METHOD PROTECTED T22_TestAddRecipeFromTemplate
VAR
	bResult: BOOL;
	sttmpLabel: ST_BaseLabel;
END_VAR
(*IF (TcUnit.TEST_ORDERED ('T22_TestAddRecipeFromTemplate')) THEN
	MEMSET (
		destAddr		:= ADR (GVL.fbRecipe.arrRecipes),
		fillByte		:= 0,
		n				:= SIZEOF (GVL.fbRecipe.arrRecipes)
	);
	WRITE_PROTECTED_UINT (ADR(GVL.fbRecipe.uiNumberOfRecipes), 0);

	
	GVL.fbRecipe.SetText (eLocation := E_BaseLocation.pl, wsDescription := "Nazwa receptury PL");
	GVL.fbRecipe.SetText (eLocation := E_BaseLocation.en, wsDescription := "Nazwa receptury EN");
	GVL.fbRecipe.SetText (eLocation := E_BaseLocation.de, wsDescription := "Nazwa receptury DE");
	

	bResult		:= GVL.fbRecipe.AddRecipeFromTemplate (uiNumberTemplates := 1, stTexts := GVL.fbRecipe.GetTexts ());	

	AssertTrue (Condition := bResult, Message := 'Test 01 - Blad utworzenia receptury');
	AssertEquals_UINT (Expected := 1, Actual := GVL.fbRecipe.GetNumberOfRecipe (), Message := 'Test 02 - Blad ilosci dodanych receptur');
	
	sttmpLabel 			:= GVL.fbRecipe.GetNamesOfRecipe (uiNumber := 1);
	AssertEquals_WSTRING (Expected := "Nazwa receptury PL", Actual := sttmpLabel.arrText [E_BaseLocation.pl], Message := 'Test 03 - bledna nazwa receptury');

	AssertEquals_UINT (Expected := 3, Actual := GVL.fbRecipe.GetNumberIngredientOfRecipe (uiNumer := 1), Message := 'Test 04 - Blad ilosci dodanych skladnikow');
	AssertEquals_WSTRING (Expected := "Nazwa skladnika 1 PL", Actual := GVL.fbRecipe.arrRecipes [1].arrIngredient [1].stTexts.arrText [1],	Message := 'Test 05 - bledna etykieta');
	AssertEquals_REAL (Expected := 1111, Actual := GVL.fbRecipe.arrRecipes [1].arrIngredient [1].rValue, 						Message := 'Test 06 - bledna wartosc', Delta := 0);
	AssertEquals_REAL (Expected := 1111, Actual := GVL.fbRecipe.arrRecipes [1].arrIngredient [1].rDefaultValue, 				Message := 'Test 07 - bledna wartosc domyslna', Delta := 0);
	AssertEquals_REAL (Expected := 1, Actual := GVL.fbRecipe.arrRecipes [1].arrIngredient [1].rMin, 							Message := 'Test 08 - bledna wartosc min', Delta := 0);
	AssertEquals_REAL (Expected := 10000, Actual := GVL.fbRecipe.arrRecipes [1].arrIngredient [1].rMax, 						Message := 'Test 09 - bledna wartosc max', Delta := 0);
	AssertEquals_WSTRING (Expected := "mm", Actual := TO_WSTRING (GVL.fbRecipe.arrRecipes [1].arrIngredient [1].sUnit), 		Message := 'Test 10 - bledna jednostka');

	TcUnit.TEST_FINISHED ();

END_IF
*)
END_METHOD

METHOD PUBLIC T23_TestDeleteRecipe
VAR
	bresult			: BOOL;
	sttmpLabel: ST_BaseLabel;
END_VAR
(*
IF (TcUnit.TEST_ORDERED ('T23_TestDeleteRecipe')) THEN
	bresult	:= GVL.fbRecipe.DeleteRecipe (uiNumber	:= 1);
	AssertTrue (Condition := bresult, Message := 'Test 01 - Bladna wynik usuwania receptury');
	AssertEquals_UINT (Expected := 0, Actual := GVL.fbRecipe.GetNumberOfRecipe (), Message := 'Test 02 - bledna ilosc receptur');

	GVL.fbRecipe.SetText (eLocation := E_BaseLocation.pl, wsDescription := "Nazwa receptury 1 PL");
	GVL.fbRecipe.SetText (eLocation := E_BaseLocation.en, wsDescription := "Nazwa receptury 1 EN");
	GVL.fbRecipe.SetText (eLocation := E_BaseLocation.de, wsDescription := "Nazwa receptury 1 DE");
	bresult := GVL.fbRecipe.AddRecipeFromTemplate (uiNumberTemplates := 1, stTexts := GVL.fbRecipe.GetTexts ());
	AssertTrue (Condition := bresult, Message := 'Test 03a - Blad dodania receptury');
	AssertEquals_UINT (Expected := 1, Actual := GVL.fbRecipe.GetNumberOfRecipe (), Message := 'Test 20a - bledna ilosc receptur');
	
	GVL.fbRecipe.SetText (eLocation := E_BaseLocation.pl, wsDescription := "Nazwa receptury 2 PL");
	GVL.fbRecipe.SetText (eLocation := E_BaseLocation.en, wsDescription := "Nazwa receptury 2 EN");
	GVL.fbRecipe.SetText (eLocation := E_BaseLocation.de, wsDescription := "Nazwa receptury 2 DE");
	bresult := GVL.fbRecipe.AddRecipeFromTemplate (uiNumberTemplates := 1, stTexts := GVL.fbRecipe.GetTexts ());
	AssertTrue (Condition := bresult, Message := 'Test 03b - Blad dodania receptury');
	AssertEquals_UINT (Expected := 2, Actual := GVL.fbRecipe.GetNumberOfRecipe (), Message := 'Test 20b - bledna ilosc receptur');

	GVL.fbRecipe.SetText (eLocation := E_BaseLocation.pl, wsDescription := "Nazwa receptury 3 PL");
	GVL.fbRecipe.SetText (eLocation := E_BaseLocation.en, wsDescription := "Nazwa receptury 3 EN");
	GVL.fbRecipe.SetText (eLocation := E_BaseLocation.de, wsDescription := "Nazwa receptury 3 DE");
	bresult := GVL.fbRecipe.AddRecipeFromTemplate (uiNumberTemplates := 1, stTexts := GVL.fbRecipe.GetTexts ());
	AssertTrue (Condition := bresult, Message := 'Test 03c - Blad dodania receptury');
	AssertEquals_UINT (Expected := 3, Actual := GVL.fbRecipe.GetNumberOfRecipe (), Message := 'Test 20c - bledna ilosc receptur');

	GVL.fbRecipe.SetText (eLocation := E_BaseLocation.pl, wsDescription := "Nazwa receptury 4 PL");
	GVL.fbRecipe.SetText (eLocation := E_BaseLocation.en, wsDescription := "Nazwa receptury 4 EN");
	GVL.fbRecipe.SetText (eLocation := E_BaseLocation.de, wsDescription := "Nazwa receptury 4 DE");
	bresult := GVL.fbRecipe.AddRecipeFromTemplate (uiNumberTemplates := 1, stTexts := GVL.fbRecipe.GetTexts ());
	AssertTrue (Condition := bresult, Message := 'Test 03d - Blad dodania receptury');
	AssertEquals_UINT (Expected := 4, Actual := GVL.fbRecipe.GetNumberOfRecipe (), Message := 'Test 20d - bledna ilosc receptur');

	bresult	:= GVL.fbRecipe.DeleteRecipe (uiNumber	:= 2);
	AssertTrue (Condition := bresult, Message := 'Test 07 - Bladna wynik usuwania receptury');
	AssertEquals_UINT (Expected := 3, Actual := GVL.fbRecipe.GetNumberOfRecipe (), Message := 'Test 08 - bledna ilosc receptur');

	sttmpLabel 			:= GVL.fbRecipe.GetNamesOfRecipe (uiNumber := 2);
	AssertEquals_WSTRING (Expected := "Nazwa receptury 3 PL", Actual := sttmpLabel.arrText [E_BaseLocation.pl], Message := 'Test 09a - bledna nazwa receptury');
	sttmpLabel 			:= GVL.fbRecipe.GetNamesOfRecipe (uiNumber := 3);
	AssertEquals_WSTRING (Expected := "Nazwa receptury 4 PL", Actual := sttmpLabel.arrText [E_BaseLocation.pl], Message := 'Test 09b - bledna nazwa receptury');
	
	TcUnit.TEST_FINISHED ();
END_IF
*)
END_METHOD

METHOD PROTECTED T24_TestCopyRecipeToNewRecipe
VAR
	bresult		: BOOL;
	sttmpLabel: ST_BaseLabel;
END_VAR
(*
IF (TcUnit.TEST_ORDERED ('T24_TestCopyRecipeToNewRecipe')) THEN
	GVL.fbRecipe.SetText (eLocation := E_BaseLocation.pl, wsDescription	:= "Nazwa receptury klon PL");
	GVL.fbRecipe.SetText (eLocation := E_BaseLocation.en, wsDescription	:= "Nazwa receptury klon EN");
	GVL.fbRecipe.SetText (eLocation := E_BaseLocation.de, wsDescription	:= "Nazwa receptury klon DE");
	

	bresult		:= GVL.fbRecipe.AddRecipeFromRecipe (uiNumberRecipe := 1, stTexts := GVL.fbRecipe.GetTexts ());	

	AssertTrue (Condition := bresult, Message := 'Test 01 - Blad utworzenia receptury');
	AssertEquals_UINT (Expected := 4, Actual := GVL.fbRecipe.GetNumberOfRecipe (), Message := 'Test 02 - Blad ilosci dodanych receptur');
	sttmpLabel 			:= GVL.fbRecipe.GetNamesOfRecipe (uiNumber := 4);
	AssertEquals_WSTRING (Expected := "Nazwa receptury klon PL", Actual := sttmpLabel.arrText [E_BaseLocation.pl], Message := 'Test 03 - bledna nazwa receptury');

	AssertEquals_UINT (Expected := 3, Actual := GVL.fbRecipe.GetNumberIngredientOfRecipe (uiNumer := 1), Message := 'Test 04 - Blad ilosci dodanych skladnikow');
	AssertEquals_WSTRING (Expected := "Nazwa skladnika 1 PL", Actual := GVL.fbRecipe.arrRecipes [4].arrIngredient [1].stTexts.arrText [1], 	Message := 'Test 05 - bledna etykieta');
	AssertEquals_REAL (Expected := 1111, Actual := GVL.fbRecipe.arrRecipes [4].arrIngredient [1].rValue, 							Message := 'Test 06 - bledna wartosc', Delta := 0);
	AssertEquals_REAL (Expected := 1111, Actual := GVL.fbRecipe.arrRecipes [4].arrIngredient [1].rDefaultValue, 					Message := 'Test 07 - bledna wartosc domyslna', Delta := 0);
	AssertEquals_REAL (Expected := 1, Actual := GVL.fbRecipe.arrRecipes [4].arrIngredient [1].rMIN, 								Message := 'Test 08 - bledna wartosc min', Delta := 0);
	AssertEquals_REAL (Expected := 10000, Actual := GVL.fbRecipe.arrRecipes [4].arrIngredient [1].rMAX, 							Message := 'Test 09 - bledna wartosc max', Delta := 0);
	AssertEquals_WSTRING (Expected := "mm", Actual := TO_WSTRING (GVL.fbRecipe.arrRecipes [4].arrIngredient [1].sUnit),			Message := 'Test 10 - bledna jednostka');

	
	TcUnit.TEST_FINISHED ();
END_IF
*)
END_METHOD

METHOD INTERNAL T99_Test
VAR_INST
	bFinish	: BOOL;
	bT99Test: BOOL;
END_VAR
(*
IF (TcUnit.TEST_ORDERED ('T99_Test')) THEN
	bT99Test			:= TRUE;

	GVL_Variable.fbPB1.ExecuteEveryCycle_Test ();
	GVL_Variable.fbPB1.ExecuteEveryCycle_Operation ();
	GVL_Variable.fbPB1.ExecuteEveryCycle_Status ();
	GVL_Variable.fbPB1.ExecuteEveryCycle_Error ();
	
	IF bFinish THEN
		bT99Test		:= FALSE;
		TcUnit.TEST_FINISHED ();
	END_IF
END_IF
*)
END_METHOD

END_FUNCTION_BLOCK

// ---- POUs/A4_Component/FB_Component.TcPOU
FUNCTION_BLOCK FB_Component EXTENDS FB_BaseComponent IMPLEMENTS ITF_Component, ITF_Component_HMI_Init
VAR
	bSetAlarm		: BOOL;
	bSetError1		: BOOL;
	bSetError2		: BOOL;
	bResetAlarm		: BOOL;
	bResetError1	: BOOL;
	bResetError2	: BOOL;
	bAckAlarm		: BOOL;
	bAckError1		: BOOL;
	bAckError2		: BOOL;

	bSetAlarm2		: BOOL;
	bSetError3		: BOOL;
	bSetError4		: BOOL;
	bResetAlarm2	: BOOL;
	bResetError3	: BOOL;
	bResetError4	: BOOL;
	bAckAlarm2		: BOOL;
	bAckError3		: BOOL;
	bAckError4		: BOOL;
	
END_VAR

IF (bSetAlarm) THEN
	bSetAlarm		:= FALSE;
	THIS^.EventSetActive (iNumber := 1);
END_IF
IF (bSetError1) THEN
	bSetError1		:= FALSE;
	THIS^.EventSetActive (iNumber := 2);
END_IF
IF (bSetError2) THEN
	bSetError2		:= FALSE;
	THIS^.EventSetActive (iNumber := 3);
END_IF
//
IF (bResetAlarm) THEN
	bResetAlarm		:= FALSE;
	THIS^.EventSetInactive (iNumber := 1);
END_IF
IF (bResetError1) THEN
	bResetError1		:= FALSE;
	THIS^.EventSetInactive (iNumber := 2);
END_IF
IF (bResetError2) THEN
	bResetError2		:= FALSE;
	THIS^.EventSetInactive (iNumber := 3);
END_IF
//
IF (bAckAlarm) THEN
	bAckAlarm		:= FALSE;
	THIS^.EventAcknowledge (iNumber := 1);
END_IF
IF (bAckError1) THEN
	bAckError1		:= FALSE;
	THIS^.EventAcknowledge (iNumber := 2);
END_IF
IF (bAckError2) THEN
	bAckError2		:= FALSE;
	THIS^.EventAcknowledge (iNumber := 3);
END_IF


IF (bSetAlarm2) THEN
	bSetAlarm2		:= FALSE;
	THIS^.EventSetActive (iNumber := 4);
END_IF
IF (bSetError3) THEN
	bSetError3		:= FALSE;
	THIS^.EventSetActive (iNumber := 5);
END_IF
IF (bSetError4) THEN
	bSetError4		:= FALSE;
	THIS^.EventSetActive (iNumber := 6);
END_IF
//
IF (bResetAlarm2) THEN
	bResetAlarm2		:= FALSE;
	THIS^.EventSetInactive (iNumber := 4);
END_IF
IF (bResetError3) THEN
	bResetError3		:= FALSE;
	THIS^.EventSetInactive (iNumber := 5);
END_IF
IF (bResetError4) THEN
	bResetError4		:= FALSE;
	THIS^.EventSetInactive (iNumber := 6);
END_IF
//
IF (bAckAlarm2) THEN
	bAckAlarm2		:= FALSE;
	THIS^.EventAcknowledge (iNumber := 4);
END_IF
IF (bAckError3) THEN
	bAckError3		:= FALSE;
	THIS^.EventAcknowledge (iNumber := 5);
END_IF
IF (bAckError4) THEN
	bAckError4		:= FALSE;
	THIS^.EventAcknowledge (iNumber := 6);
END_IF

(*			
	EVERDE sp. z o.o.
	Rafał Osajda		24.03.2025		TC 4024.66
	Definicja nowego zgłoszenia
*)
METHOD PUBLIC EventsDefinition : BOOL
VAR
	fbName					: FB_BaseLabel;
END_VAR
SUPER^.EventsDefinition ();

fbName.SetText (eLocation := E_BaseLocation.pl, wsDescription := "Zgloszneie komponentu 1 PL");
fbName.SetText (eLocation := E_BaseLocation.en, wsDescription := "Zgloszneie komponentu 1 EN");
fbName.SetText (eLocation := E_BaseLocation.de, wsDescription := "Zgloszneie komponentu 1 DE");
THIS^.AddEvent (
	bIgnoreRepetitions		:= TRUE,
	eEventCategory			:= E_BaseEvents_Category.ALARM,
	bConfirm				:= FALSE,
	stDescription			:= fbName.GetTexts ()
);

fbName.SetText (eLocation := E_BaseLocation.pl, wsDescription := "Zgloszneie komponentu 2 PL");
fbName.SetText (eLocation := E_BaseLocation.en, wsDescription := "Zgloszneie komponentu 2 EN");
fbName.SetText (eLocation := E_BaseLocation.de, wsDescription := "Zgloszneie komponentu 2 DE");
THIS^.AddEvent (
	bIgnoreRepetitions		:= TRUE,
	eEventCategory			:= E_BaseEvents_Category.Error,
	bConfirm				:= FALSE,
	stDescription			:= fbName.GetTexts ()
);

fbName.SetText (eLocation := E_BaseLocation.pl, wsDescription := "Zgloszneie komponentu 3 PL");
fbName.SetText (eLocation := E_BaseLocation.en, wsDescription := "Zgloszneie komponentu 3 EN");
fbName.SetText (eLocation := E_BaseLocation.de, wsDescription := "Zgloszneie komponentu 3 DE");
THIS^.AddEvent (
	bIgnoreRepetitions		:= TRUE,
	eEventCategory			:= E_BaseEvents_Category.Error,
	bConfirm				:= TRUE,
	stDescription			:= fbName.GetTexts ()
);

fbName.SetText (eLocation := E_BaseLocation.pl, wsDescription := "Zgloszneie komponentu 4 PL");
fbName.SetText (eLocation := E_BaseLocation.en, wsDescription := "Zgloszneie komponentu 4 EN");
fbName.SetText (eLocation := E_BaseLocation.de, wsDescription := "Zgloszneie komponentu 4 DE");
THIS^.AddEvent (
	bIgnoreRepetitions		:= TRUE,
	eEventCategory			:= E_BaseEvents_Category.ALARM,
	bConfirm				:= FALSE,
	stDescription			:= fbName.GetTexts ()
);

fbName.SetText (eLocation := E_BaseLocation.pl, wsDescription := "Zgloszneie komponentu 5 PL");
fbName.SetText (eLocation := E_BaseLocation.en, wsDescription := "Zgloszneie komponentu 5 EN");
fbName.SetText (eLocation := E_BaseLocation.de, wsDescription := "Zgloszneie komponentu 5 DE");
THIS^.AddEvent (
	bIgnoreRepetitions		:= TRUE,
	eEventCategory			:= E_BaseEvents_Category.Error,
	bConfirm				:= FALSE,
	stDescription			:= fbName.GetTexts ()
);

fbName.SetText (eLocation := E_BaseLocation.pl, wsDescription := "Zgloszneie komponentu 6 PL");
fbName.SetText (eLocation := E_BaseLocation.en, wsDescription := "Zgloszneie komponentu 6 EN");
fbName.SetText (eLocation := E_BaseLocation.de, wsDescription := "Zgloszneie komponentu 6 DE");
THIS^.AddEvent (
	bIgnoreRepetitions		:= TRUE,
	eEventCategory			:= E_BaseEvents_Category.Error,
	bConfirm				:= TRUE,
	stDescription			:= fbName.GetTexts ()
);
END_METHOD

END_FUNCTION_BLOCK

// ---- POUs/A5_ControlElement_1/FB_ControlElement_1.TcPOU
FUNCTION_BLOCK FB_ControlElement_1 EXTENDS FB_BaseControlElement IMPLEMENTS ITF_ControlElement_1, ITF_ControlElement_HMI_Init
VAR
	itfComponent1				: ITF_Component;
	itfComponent2				: ITF_Component;
	
	bHomingFinished				: BOOL;
END_VAR

(*			
	EVERDE sp. z o.o.
	Rafał Osajda		24.03.2025		TC 4024.66
	Definicja nowego zgłoszenia
*)
METHOD PUBLIC EventsDefinition : BOOL
VAR
	fbName					: FB_BaseLabel;
END_VAR
SUPER^.EventsDefinition ();

fbName.SetText (eLocation := E_BaseLocation.pl, wsDescription := "Zgloszneie Wykonawczego 1 PL");
fbName.SetText (eLocation := E_BaseLocation.en, wsDescription := "Zgloszneie Wykonawczego 1 EN");
fbName.SetText (eLocation := E_BaseLocation.de, wsDescription := "Zgloszneie Wykonawczego 1 DE");
THIS^.AddEvent (
	bIgnoreRepetitions		:= TRUE,
	eEventCategory			:= E_BaseEvents_Category.ALARM,
	bConfirm				:= FALSE,
	stDescription			:= fbName.GetTexts ()
);

fbName.SetText (eLocation := E_BaseLocation.pl, wsDescription := "Zgloszneie Wykonawczego 2 PL");
fbName.SetText (eLocation := E_BaseLocation.en, wsDescription := "Zgloszneie Wykonawczego 2 EN");
fbName.SetText (eLocation := E_BaseLocation.de, wsDescription := "Zgloszneie Wykonawczego 2 DE");
THIS^.AddEvent (
	bIgnoreRepetitions		:= TRUE,
	eEventCategory			:= E_BaseEvents_Category.ALARM,
	bConfirm				:= FALSE,
	stDescription			:= fbName.GetTexts ()
);

fbName.SetText (eLocation := E_BaseLocation.pl, wsDescription := "Zgloszneie Wykonawczego 3 PL");
fbName.SetText (eLocation := E_BaseLocation.en, wsDescription := "Zgloszneie Wykonawczego 3 EN");
fbName.SetText (eLocation := E_BaseLocation.de, wsDescription := "Zgloszneie Wykonawczego 3 DE");
THIS^.AddEvent (
	bIgnoreRepetitions		:= TRUE,
	eEventCategory			:= E_BaseEvents_Category.ALARM,
	bConfirm				:= FALSE,
	stDescription			:= fbName.GetTexts ()
);
END_METHOD

METHOD FB_init : BOOL
VAR_INPUT
	bInitRetains : BOOL; // if TRUE, the retain variables are initialized (warm start / cold start)
	bInCopyCode : BOOL;  // if TRUE, the instance afterwards gets moved into the copy code (online change)
	itfComponent1				: ITF_Component;
	itfComponent2				: ITF_Component;
END_VAR
THIS^.itfComponent1					:= itfComponent1;
THIS^.AddComponent (itfComponent	:= itfComponent1);
THIS^.SetText (eLocation 			:= E_BaseLocation.pl, wsDescription := "Nazwa komponentu 1 pl");
THIS^.SetText (eLocation 			:= E_BaseLocation.en, wsDescription := "Nazwa komponentu 1 en");
THIS^.SetText (eLocation 			:= E_BaseLocation.de, wsDescription := "Nazwa komponentu 1 de");
THIS^.itfComponent1.SetName (stName	:= THIS^.GetTexts ());

THIS^.itfComponent2					:= itfComponent2;
THIS^.AddComponent (itfComponent	:= itfComponent2);
THIS^.SetText (eLocation 			:= E_BaseLocation.pl, wsDescription := "Nazwa komponentu 2 pl");
THIS^.SetText (eLocation 			:= E_BaseLocation.en, wsDescription := "Nazwa komponentu 2 en");
THIS^.SetText (eLocation 			:= E_BaseLocation.de, wsDescription := "Nazwa komponentu 2 de");
THIS^.itfComponent2.SetName (stName	:= THIS^.GetTexts ());
END_METHOD

(*			
	EVERDE sp. z o.o.
	Rafał Osajda		27.05.2025		TC 4024.66
	Metoda bazowania kontrektnego elementu 
*)
METHOD PROTECTED HomingCycle : BOOL
VAR_INPUT
END_VAR
CASE THIS^.stHoming.iChildHomingStep OF
0	:
	IF (THIS^.bHomingFinished) THEN
		THIS^.bHomingFinished		:= FALSE;
		THIS^.stHoming.iChildHomingStep	:= 10;
	END_IF
	HomingCycle					:= TRUE;
10	:
	this^.stHoming.iChildHomingStep	:= 0;
	HomingCycle					:= FALSE;
END_CASE
END_METHOD

END_FUNCTION_BLOCK

// ---- POUs/A4_Component/FB_Component_HMI.TcPOU
FUNCTION_BLOCK FB_Component_HMI EXTENDS FB_BaseComponent_HMI IMPLEMENTS ITF_Component_HMI
VAR
	itfComponentConnector				: ITF_Component_HMI_Connector;
	refstComponentData					: REFERENCE TO ST_Component_HMI;
	
END_VAR

METHOD FB_init : BOOL
VAR_INPUT
	bInitRetains : BOOL; // if TRUE, the retain variables are initialized (warm start / cold start)
	bInCopyCode : BOOL;  // if TRUE, the instance afterwards gets moved into the copy code (online change)
	itfBaseLoggerConnector				: ITF_BaseLogger_HMI_Connector;	//bezpośredni łącznik do logera
	itfComponentConnector				: ITF_Component_HMI_Init;
END_VAR
//Przypisanie do elementu który własnie stworzyliśmy
THIS^.itfComponentConnector				:= itfComponentConnector;
//Przypisanie do elementów z biblioteki
THIS^.itfBaseLoggerElementConnector		:= itfComponentConnector;
THIS^.itfBaseComponentConnector			:= itfComponentConnector;

//
THIS^.itfBaseLoggerConnector			:= itfBaseLoggerConnector;

IF (THIS^.itfComponentConnector <> 0 AND
	THIS^.itfBaseLoggerElementConnector <> 0 AND
	THIS^.itfBaseComponentConnector	<> 0 AND
	THIS^.itfBaseLoggerConnector <> 0) THEN
	THIS^.bIsInit						:= TRUE;
END_IF
END_METHOD

METHOD LinkComponentData : BOOL
VAR_INPUT
	stData					: REFERENCE TO ST_Component_HMI_Link;
END_VAR
THIS^.refstComponentData	REF= stData.stComponent;

THIS^.refstBaseLoggerElementDataHMI	REF= stData.stBaseLoggerElement;
THIS^.refstBaseComponentDataHMI		REF= stData.stBaseComponent;

THIS^.CreateLinkToEventsMemory ();

IF (__ISVALIDREF (THIS^.refstComponentData) AND THIS^.IsLinkedReferences ()) THEN
	THIS^.bIsValidData		:= TRUE;
	LinkComponentData		:= TRUE;
END_IF
END_METHOD

END_FUNCTION_BLOCK

// ---- POUs/A5_ControlElement/FB_ControlElement_HMI.TcPOU
FUNCTION_BLOCK FB_ControlElement_HMI EXTENDS FB_BaseControlElement_HMI IMPLEMENTS ITF_ControlElement_HMI
VAR
	itfControlElementConnector			: ITF_ControlElement_HMI_Connector;
	refstControlElementData				: REFERENCE TO ST_ControlElement_HMI;
	
	itfComponent1						: ITF_Component_HMI;
	itfComponent2						: ITF_Component_HMI;
END_VAR

METHOD FB_init : BOOL
VAR_INPUT
	bInitRetains : BOOL; // if TRUE, the retain variables are initialized (warm start / cold start)
	bInCopyCode : BOOL;  // if TRUE, the instance afterwards gets moved into the copy code (online change)
	itfBaseLoggerConnector				: ITF_BaseLogger_HMI_Connector;	//bezpośredni łącznik do logera
	itfControlElementConnector			: ITF_ControlElement_HMI_Init;
	itfComponent1						: ITF_Component_HMI;
	itfComponent2						: ITF_Component_HMI;
END_VAR
//Przypisanie do elementu który własnie stworzyliśmy
THIS^.itfControlElementConnector		:= itfControlElementConnector;
//Przypisanie do elementów z biblioteki
THIS^.itfBaseLoggerElementConnector		:= itfControlElementConnector;
THIS^.itfBaseComponentConnector			:= itfControlElementConnector;
THIS^.itfBaseControlElementConnector	:= itfControlElementConnector;
//
THIS^.itfBaseLoggerConnector			:= itfBaseLoggerConnector;
//
THIS^.itfComponent1						:= itfComponent1;
THIS^.AddComponent (itfComponentHMI		:= itfComponent1);
THIS^.itfComponent2						:= itfComponent2;
this^.AddComponent (itfComponentHMI		:= itfComponent2);

IF (THIS^.itfControlElementConnector <> 0 AND
	THIS^.itfBaseLoggerElementConnector <> 0 AND
	THIS^.itfBaseComponentConnector	<> 0 AND
	THIS^.itfBaseControlElementConnector <> 0 AND
	THIS^.itfBaseLoggerConnector <> 0) THEN
	THIS^.bIsInit						:= TRUE;
END_IF
END_METHOD

METHOD LinkControlElementData : BOOL
VAR_INPUT
	stData				: reference to ST_ControlElement_HMI_Link;
END_VAR
THIS^.refstControlElementData			REF= stData.stControlElement;	//ta zmienna powstaje w elemencie 

THIS^.refstBaseLoggerElementDataHMI		REF= stData.stBaseLoggerElement;	//zmienne z biblioteki ale dopiero tu je moge przypisać 
THIS^.refstBaseComponentDataHMI			REF= stData.stBaseComponent;
THIS^.refstBaseControlElementDataHMI	REF= stData.stBaseControlElement;

THIS^.itfComponent1.LinkComponentData (stData := stData.stComponent1);	//przekazanie danych do elementu podrzędnego np do czujnika
THIS^.itfComponent2.LinkComponentData (stData := stData.stComponent2);

THIS^.CreateLinkToEventsMemory ();	//wywołanie metody linkującą poamięc zgłoszęń

IF (__ISVALIDREF (THIS^.refstControlElementData) AND this^.IsLinkedReferences ()) THEN
	THIS^.bIsValidData		:= TRUE;
	LinkControlElementData	:= TRUE;
END_IF
END_METHOD

END_FUNCTION_BLOCK

// ---- POUs/A0_BaseFB/Command/FB_CommandChild.TcPOU
FUNCTION_BLOCK FB_CommandChild EXTENDS FB_BaseCommand
VAR
	bFinish				: BOOL;
	iI1					: INT;
	iI2					: INT;
END_VAR

IF (THIS^.IsFirstCycle ()) THEN
	iI1 := iI1 + 1;
END_IF
IF (THIS^.IsLastCycle ()) THEN
	iI2 := iI2 + 1;
END_IF

METHOD PUBLIC CyklTestu : BOOL
VAR_INPUT
END_VAR
CASE THIS^.GetStep () OF
0	:
	THIS^.SetStepINC10 ();
10	:
	IF (THIS^.bFinish) THEN
		THIS^.SetStepAsFinal ();
	END_IF
END_CASE
CyklTestu			:= THIS^.TestingLastCycle ();
END_METHOD

END_FUNCTION_BLOCK

// ---- POUs/A2_logger/FB_LoggerTest.TcPOU
FUNCTION_BLOCK FB_LoggerTest EXTENDS TcUnit.FB_TestSuite
VAR

END_VAR


T01_TestDodawaniaZgloszen ();
T02_TestDodawaniaZgloszen2 ();
T03_TestDodawaniaZgloszen3 ();
T04_TestDodawaniaKomponentowDoLogera ();
//T05_TestDodawaniaWykonawczychDoLogera ();
//T06_TestDodawaniaZlozonychDoLogera ();
//T07_TestDodawaniaBazowychDoLogera ();

METHOD PRIVATE T01_TestDodawaniaZgloszen
VAR
	sttmpEvent: ST_BaseEvents_RowInQueue;
END_VAR
IF (TcUnit.TEST_ORDERED ('T01_TestDodawaniaZgloszen')) THEN
	WRITE_PROTECTED_BOOL (Ptr := ADR (GVL.fbLogger.bClearMemory), Value := TRUE);
	GVL.fbLogger ();
	AssertEquals_INT (Expected := 0, Actual := GVL.fbLogger.stBuffer.iNumerOfEvents, 	Message := 'T01a - bledna ilosc w kolejce');
	AssertEquals_INT (Expected := 0, Actual := GVL.fbLogger.stmemory.iNumberOfRow,		Message := 'T01b - bledna ilosc zgloszen');
//wyslanie zgloszenia 
	sttmpEvent.bActive				:= TRUE;
	sttmpEvent.bConfirm				:= TRUE;
	sttmpEvent.bIgnoreRepetitions	:= TRUE;
	sttmpEvent.dtStart				:= DT#2025-09-25-01:00:00;
	sttmpEvent.eEventCategory		:= E_BaseEvents_Category.Error;
	sttmpEvent.eEventAction			:= E_BaseEvents_Action.Start;
	sttmpEvent.uiIDEvent			:= 1;
	sttmpEvent.uiIDItem				:= 2;
	GVL.fbLogger.ReportEvent (stEvent := sttmpEvent);
	AssertEquals_INT (Expected := 1, Actual := GVL.fbLogger.stBuffer.iNumerOfEvents, 	Message := 'T02a - bledna ilosc w kolejce');
	AssertEquals_INT (Expected := 0, Actual := GVL.fbLogger.stmemory.iNumberOfRow,		Message := 'T02b - bledna ilosc zgloszen');
	GVL.fbLogger ();
	AssertEquals_INT (Expected := 0, Actual := GVL.fbLogger.stBuffer.iNumerOfEvents, 					Message := 'T03a - bledna ilosc w kolejce');
	AssertEquals_INT (Expected := 1, Actual := GVL.fbLogger.stmemory.iNumberOfRow,						Message := 'T03b - bledna ilosc zgloszen');
	AssertEquals_INT (Expected := 1, Actual := GVL.fbLogger.stNumberOfReports.iNumberOfActive,			Message := 'T03c - bledna ilosc zgloszen');
	AssertTrue (Condition := GVL.fbLogger.stNumberOfReports.arrActive [E_BaseEvents_Category.Error],	Message := 'T03d - bledny stan');
	AssertFalse (Condition := GVL.fbLogger.stNumberOfReports.arrActive [E_BaseEvents_Category.Alarm],	Message := 'T03d - bledny stan');
	AssertTrue (Condition := GVL.fbLogger.stNumberOfReports.bIsActive,									Message := 'T03e - bledny stan');
	AssertEquals_INT (Expected := 1, Actual := GVL.fbLogger.stNumberOfReports.iTotalNumer,				Message := 'T03f - bledna ilosc zgloszen');
//potwierdzenie zgloszenia 
	sttmpEvent.eEventAction			:= E_BaseEvents_Action.Confirm;
	sttmpEvent.uiIDEvent			:= 1;
	sttmpEvent.uiIDItem				:= 2;
	sttmpEvent.dtConfirmed			:= DT#2025-09-25-01:01:00;
	GVL.fbLogger.ReportEvent (stEvent := sttmpEvent);
	AssertEquals_INT (Expected := 1, Actual := GVL.fbLogger.stBuffer.iNumerOfEvents, 					Message := 'T04a - bledna ilosc w kolejce');
	AssertEquals_INT (Expected := 1, Actual := GVL.fbLogger.stmemory.iNumberOfRow,						Message := 'T04b - bledna ilosc zgloszen');
	GVL.fbLogger ();
	AssertEquals_INT (Expected := 0, Actual := GVL.fbLogger.stBuffer.iNumerOfEvents, 					Message := 'T05a - bledna ilosc w kolejce');
	AssertEquals_INT (Expected := 1, Actual := GVL.fbLogger.stmemory.iNumberOfRow,						Message := 'T05b - bledna ilosc zgloszen');
	AssertEquals_INT (Expected := 1, Actual := GVL.fbLogger.stNumberOfReports.iNumberOfActive,			Message := 'T05c - bledna ilosc zgloszen');
	AssertTrue (Condition := GVL.fbLogger.stNumberOfReports.arrActive [E_BaseEvents_Category.Error],	Message := 'T05d - bledny stan');
	AssertFalse (Condition := GVL.fbLogger.stNumberOfReports.arrActive [E_BaseEvents_Category.Alarm],	Message := 'T05d - bledny stan');
	AssertTrue (Condition := GVL.fbLogger.stNumberOfReports.bIsActive,									Message := 'T05e - bledny stan');
	AssertEquals_INT (Expected := 1, Actual := GVL.fbLogger.stNumberOfReports.iTotalNumer,				Message := 'T05f - bledna ilosc zgloszen');
//zamkniecie zgloszenia 
	sttmpEvent.eEventAction			:= E_BaseEvents_Action.Stop;
	sttmpEvent.uiIDEvent			:= 1;
	sttmpEvent.uiIDItem				:= 2;
	sttmpEvent.dtFinish				:= DT#2025-09-25-01:02:00;
	GVL.fbLogger.ReportEvent (stEvent := sttmpEvent);
	AssertEquals_INT (Expected := 1, Actual := GVL.fbLogger.stBuffer.iNumerOfEvents, 					Message := 'T04a - bledna ilosc w kolejce');
	AssertEquals_INT (Expected := 1, Actual := GVL.fbLogger.stmemory.iNumberOfRow,						Message := 'T04b - bledna ilosc zgloszen');
	GVL.fbLogger ();
	AssertEquals_INT (Expected := 0, Actual := GVL.fbLogger.stBuffer.iNumerOfEvents, 					Message := 'T05a - bledna ilosc w kolejce');
	AssertEquals_INT (Expected := 1, Actual := GVL.fbLogger.stmemory.iNumberOfRow,						Message := 'T05b - bledna ilosc zgloszen');
	AssertEquals_INT (Expected := 0, Actual := GVL.fbLogger.stNumberOfReports.iNumberOfActive,			Message := 'T05c - bledna ilosc zgloszen');
	AssertFalse (Condition := GVL.fbLogger.stNumberOfReports.arrActive [E_BaseEvents_Category.Error],	Message := 'T05d - bledny stan');
	AssertFalse (Condition := GVL.fbLogger.stNumberOfReports.arrActive [E_BaseEvents_Category.Alarm],	Message := 'T05d - bledny stan');
	Assertfalse (Condition := GVL.fbLogger.stNumberOfReports.bIsActive,									Message := 'T05e - bledny stan');
	AssertEquals_INT (Expected := 1, Actual := GVL.fbLogger.stNumberOfReports.iTotalNumer,				Message := 'T05f - bledna ilosc zgloszen');
	
	
	TcUnit.TEST_FINISHED ();
END_IF
END_METHOD

METHOD PRIVATE T02_TestDodawaniaZgloszen2
VAR
	sttmpEvent: ST_BaseEvents_RowInQueue;
END_VAR
IF (TcUnit.TEST_ORDERED ('T02_TestDodawaniaZgloszen2')) THEN
	GVL.fbLogger ();
	AssertEquals_INT (Expected := 0, Actual := GVL.fbLogger.stBuffer.iNumerOfEvents, 	Message := 'T01a - bledna ilosc w kolejce');
	AssertEquals_INT (Expected := 1, Actual := GVL.fbLogger.stmemory.iNumberOfRow,		Message := 'T01b - bledna ilosc zgloszen');
//wyslanie zgloszenia 
	sttmpEvent.bActive				:= TRUE;
	sttmpEvent.bConfirm				:= TRUE;
	sttmpEvent.bIgnoreRepetitions	:= TRUE;
	sttmpEvent.dtStart				:= DT#2025-09-25-02:00:00;
	sttmpEvent.eEventCategory		:= E_BaseEvents_Category.Error;
	sttmpEvent.eEventAction			:= E_BaseEvents_Action.Start;
	sttmpEvent.uiIDEvent			:= 1;
	sttmpEvent.uiIDItem				:= 2;
	GVL.fbLogger.ReportEvent (stEvent := sttmpEvent);
	AssertEquals_INT (Expected := 1, Actual := GVL.fbLogger.stBuffer.iNumerOfEvents, 					Message := 'T02a - bledna ilosc w kolejce');
	AssertEquals_INT (Expected := 1, Actual := GVL.fbLogger.stmemory.iNumberOfRow,						Message := 'T02b - bledna ilosc zgloszen');
	GVL.fbLogger ();
	AssertEquals_INT (Expected := 0, Actual := GVL.fbLogger.stBuffer.iNumerOfEvents, 					Message := 'T03a - bledna ilosc w kolejce');
	AssertEquals_INT (Expected := 2, Actual := GVL.fbLogger.stmemory.iNumberOfRow,						Message := 'T03b - bledna ilosc zgloszen');
	AssertEquals_INT (Expected := 1, Actual := GVL.fbLogger.stNumberOfReports.iNumberOfActive,			Message := 'T03c - bledna ilosc zgloszen');
	AssertTrue (Condition := GVL.fbLogger.stNumberOfReports.arrActive [E_BaseEvents_Category.Error],	Message := 'T03d - bledny stan');
	AssertFalse (Condition := GVL.fbLogger.stNumberOfReports.arrActive [E_BaseEvents_Category.Alarm],	Message := 'T03d - bledny stan');
	AssertTrue (Condition := GVL.fbLogger.stNumberOfReports.bIsActive,									Message := 'T03e - bledny stan');
	AssertEquals_INT (Expected := 2, Actual := GVL.fbLogger.stNumberOfReports.iTotalNumer,				Message := 'T03f - bledna ilosc zgloszen');
//zamkniecie zgloszenia  bez potwierdzenia a wymagane nic się nei powinno stać
	sttmpEvent.eEventAction			:= E_BaseEvents_Action.Stop;
	sttmpEvent.uiIDEvent			:= 1;
	sttmpEvent.uiIDItem				:= 2;
	sttmpEvent.dtFinish				:= DT#2025-09-25-02:00:00;
	GVL.fbLogger.ReportEvent (stEvent := sttmpEvent);
	AssertEquals_INT (Expected := 1, Actual := GVL.fbLogger.stBuffer.iNumerOfEvents, 					Message := 'T04a - bledna ilosc w kolejce');
	AssertEquals_INT (Expected := 2, Actual := GVL.fbLogger.stmemory.iNumberOfRow,						Message := 'T04b - bledna ilosc zgloszen');
	GVL.fbLogger ();
	AssertEquals_INT (Expected := 0, Actual := GVL.fbLogger.stBuffer.iNumerOfEvents, 					Message := 'T05a - bledna ilosc w kolejce');
	AssertEquals_INT (Expected := 2, Actual := GVL.fbLogger.stmemory.iNumberOfRow,						Message := 'T05b - bledna ilosc zgloszen');
	AssertEquals_INT (Expected := 1, Actual := GVL.fbLogger.stNumberOfReports.iNumberOfActive,			Message := 'T05c - bledna ilosc zgloszen');
	AssertTrue (Condition := GVL.fbLogger.stNumberOfReports.arrActive [E_BaseEvents_Category.Error],	Message := 'T05d - bledny stan');
	AssertFalse (Condition := GVL.fbLogger.stNumberOfReports.arrActive [E_BaseEvents_Category.Alarm],	Message := 'T05d - bledny stan');
	AssertTrue (Condition := GVL.fbLogger.stNumberOfReports.bIsActive,									Message := 'T05e - bledny stan');
	AssertEquals_INT (Expected := 2, Actual := GVL.fbLogger.stNumberOfReports.iTotalNumer,				Message := 'T05f - bledna ilosc zgloszen');
//potwierdzenie zgloszenia 
	sttmpEvent.eEventAction			:= E_BaseEvents_Action.Confirm;
	sttmpEvent.uiIDEvent			:= 1;
	sttmpEvent.uiIDItem				:= 2;
	sttmpEvent.dtConfirmed			:= DT#2025-09-25-02:01:00;
	GVL.fbLogger.ReportEvent (stEvent := sttmpEvent);
	AssertEquals_INT (Expected := 1, Actual := GVL.fbLogger.stBuffer.iNumerOfEvents, 					Message := 'T06a - bledna ilosc w kolejce');
	AssertEquals_INT (Expected := 2, Actual := GVL.fbLogger.stmemory.iNumberOfRow,						Message := 'T06b - bledna ilosc zgloszen');
	GVL.fbLogger ();
	AssertEquals_INT (Expected := 0, Actual := GVL.fbLogger.stBuffer.iNumerOfEvents, 					Message := 'T07a - bledna ilosc w kolejce');
	AssertEquals_INT (Expected := 2, Actual := GVL.fbLogger.stmemory.iNumberOfRow,						Message := 'T07b - bledna ilosc zgloszen');
	AssertEquals_INT (Expected := 1, Actual := GVL.fbLogger.stNumberOfReports.iNumberOfActive,			Message := 'T07c - bledna ilosc zgloszen');
	AssertTrue (Condition := GVL.fbLogger.stNumberOfReports.arrActive [E_BaseEvents_Category.Error],	Message := 'T07d - bledny stan');
	AssertFalse (Condition := GVL.fbLogger.stNumberOfReports.arrActive [E_BaseEvents_Category.Alarm],	Message := 'T07d - bledny stan');
	AssertTrue (Condition := GVL.fbLogger.stNumberOfReports.bIsActive,									Message := 'T07e - bledny stan');
	AssertEquals_INT (Expected := 2, Actual := GVL.fbLogger.stNumberOfReports.iTotalNumer,				Message := 'T07f - bledna ilosc zgloszen');
//zamkniecie zgloszenia 
	sttmpEvent.eEventAction			:= E_BaseEvents_Action.Stop;
	sttmpEvent.uiIDEvent			:= 1;
	sttmpEvent.uiIDItem				:= 2;
	sttmpEvent.dtFinish				:= DT#2025-09-25-02:02:00;
	GVL.fbLogger.ReportEvent (stEvent := sttmpEvent);
	AssertEquals_INT (Expected := 1, Actual := GVL.fbLogger.stBuffer.iNumerOfEvents, 					Message := 'T08a - bledna ilosc w kolejce');
	AssertEquals_INT (Expected := 2, Actual := GVL.fbLogger.stmemory.iNumberOfRow,						Message := 'T08b - bledna ilosc zgloszen');
	GVL.fbLogger ();
	AssertEquals_INT (Expected := 0, Actual := GVL.fbLogger.stBuffer.iNumerOfEvents, 					Message := 'T09a - bledna ilosc w kolejce');
	AssertEquals_INT (Expected := 2, Actual := GVL.fbLogger.stmemory.iNumberOfRow,						Message := 'T09b - bledna ilosc zgloszen');
	AssertEquals_INT (Expected := 0, Actual := GVL.fbLogger.stNumberOfReports.iNumberOfActive,			Message := 'T09c - bledna ilosc zgloszen');
	AssertFalse (Condition := GVL.fbLogger.stNumberOfReports.arrActive [E_BaseEvents_Category.Error],	Message := 'T09d - bledny stan');
	AssertFalse (Condition := GVL.fbLogger.stNumberOfReports.arrActive [E_BaseEvents_Category.Alarm],	Message := 'T09d - bledny stan');
	Assertfalse (Condition := GVL.fbLogger.stNumberOfReports.bIsActive,									Message := 'T09e - bledny stan');
	AssertEquals_INT (Expected := 2, Actual := GVL.fbLogger.stNumberOfReports.iTotalNumer,				Message := 'T09f - bledna ilosc zgloszen');
	
	
	TcUnit.TEST_FINISHED ();
END_IF
END_METHOD

METHOD PRIVATE T03_TestDodawaniaZgloszen3
VAR
	sttmpEvent: ST_BaseEvents_RowInQueue;
END_VAR
IF (TcUnit.TEST_ORDERED ('T03_TestDodawaniaZgloszen3')) THEN
//wyslanie zgloszenia 
	sttmpEvent.bActive				:= TRUE;
	sttmpEvent.bConfirm				:= FALSE;
	sttmpEvent.bIgnoreRepetitions	:= FALSE;
	sttmpEvent.dtStart				:= DT#2025-09-25-03:00:00;
	sttmpEvent.eEventCategory		:= E_BaseEvents_Category.Alarm;
	sttmpEvent.eEventAction			:= E_BaseEvents_Action.Start;
	sttmpEvent.uiIDEvent			:= 1;
	sttmpEvent.uiIDItem				:= 1;
	GVL.fbLogger.ReportEvent (stEvent := sttmpEvent);
	GVL.fbLogger ();
//zamkniecie zgloszenia 
	sttmpEvent.eEventAction			:= E_BaseEvents_Action.Stop;
	sttmpEvent.uiIDEvent			:= 1;
	sttmpEvent.uiIDItem				:= 1;
	sttmpEvent.dtFinish				:= DT#2025-09-25-03:02:00;
	GVL.fbLogger.ReportEvent (stEvent := sttmpEvent);
	GVL.fbLogger ();
//wyslanie zgloszenia 
	sttmpEvent.bActive				:= TRUE;
	sttmpEvent.bConfirm				:= FALSE;
	sttmpEvent.bIgnoreRepetitions	:= FALSE;
	sttmpEvent.dtStart				:= DT#2025-09-25-03:10:00;
	sttmpEvent.eEventCategory		:= E_BaseEvents_Category.Alarm;
	sttmpEvent.eEventAction			:= E_BaseEvents_Action.Start;
	sttmpEvent.uiIDEvent			:= 1;
	sttmpEvent.uiIDItem				:= 1;
	GVL.fbLogger.ReportEvent (stEvent := sttmpEvent);
	GVL.fbLogger ();
//wyslanie zgloszenia 
	sttmpEvent.bActive				:= TRUE;
	sttmpEvent.bConfirm				:= TRUE;
	sttmpEvent.bIgnoreRepetitions	:= TRUE;
	sttmpEvent.dtStart				:= DT#2025-09-25-03:20:00;
	sttmpEvent.eEventCategory		:= E_BaseEvents_Category.Error;
	sttmpEvent.eEventAction			:= E_BaseEvents_Action.Start;
	sttmpEvent.uiIDEvent			:= 2;
	sttmpEvent.uiIDItem				:= 1;
	GVL.fbLogger.ReportEvent (stEvent := sttmpEvent);
	GVL.fbLogger ();
//potwierdzenie zgloszenia 
	sttmpEvent.eEventAction			:= E_BaseEvents_Action.Confirm;
	sttmpEvent.uiIDEvent			:= 2;
	sttmpEvent.uiIDItem				:= 1;
	sttmpEvent.dtConfirmed			:= DT#2025-09-25-03:21:00;
	GVL.fbLogger.ReportEvent (stEvent := sttmpEvent);
	GVL.fbLogger ();
//zamkniecie zgloszenia 
	sttmpEvent.eEventAction			:= E_BaseEvents_Action.Stop;
	sttmpEvent.uiIDEvent			:= 2;
	sttmpEvent.uiIDItem				:= 1;
	sttmpEvent.dtFinish				:= DT#2025-09-25-03:22:00;
	GVL.fbLogger.ReportEvent (stEvent := sttmpEvent);
	GVL.fbLogger ();
//wyslanie zgloszenia 
	sttmpEvent.bActive				:= TRUE;
	sttmpEvent.bConfirm				:= FALSE;
	sttmpEvent.bIgnoreRepetitions	:= TRUE;
	sttmpEvent.dtStart				:= DT#2025-09-25-04:00:00;
	sttmpEvent.eEventCategory		:= E_BaseEvents_Category.Error;
	sttmpEvent.eEventAction			:= E_BaseEvents_Action.Start;
	sttmpEvent.uiIDEvent			:= 3;
	sttmpEvent.uiIDItem				:= 1;
	GVL.fbLogger.ReportEvent (stEvent := sttmpEvent);
	GVL.fbLogger ();
//wyslanie zgloszenia 
	sttmpEvent.bActive				:= TRUE;
	sttmpEvent.bConfirm				:= FALSE;
	sttmpEvent.bIgnoreRepetitions	:= TRUE;
	sttmpEvent.dtStart				:= DT#2025-09-25-04:20:00;
	sttmpEvent.eEventCategory		:= E_BaseEvents_Category.Message;
	sttmpEvent.eEventAction			:= E_BaseEvents_Action.Start;
	sttmpEvent.uiIDEvent			:= 4;
	sttmpEvent.uiIDItem				:= 1;
	GVL.fbLogger.ReportEvent (stEvent := sttmpEvent);
	GVL.fbLogger ();
//zamkniecie zgloszenia 
	sttmpEvent.eEventAction			:= E_BaseEvents_Action.Stop;
	sttmpEvent.uiIDEvent			:= 4;
	sttmpEvent.uiIDItem				:= 1;
	sttmpEvent.dtFinish				:= DT#2025-09-25-04:22:00;
	GVL.fbLogger.ReportEvent (stEvent := sttmpEvent);
	GVL.fbLogger ();
	
	
	TcUnit.TEST_FINISHED ();
END_IF
END_METHOD

METHOD PROTECTED T04_TestDodawaniaKomponentowDoLogera
VAR_INPUT
END_VAR

VAR
	iWynik: INT;
END_VAR
IF (TcUnit.TEST_ORDERED ('T04_TestDodawaniaKomponentowDoLogera')) THEN
	iWynik :=	GVL_Variable.fbComponent_1_L.SetID (uiID 	:= 1);
	iWynik :=	GVL_Variable.fbComponent_2_L.SetID (uiID 	:= TO_UINT (iWynik + 1));
	iWynik :=	GVL_Variable.fbComponent_3_L.SetID (uiID 	:= TO_UINT (iWynik + 1));

	GVL.fbLogger.AddItem (itfItem := GVL_Variable.fbComponent_1_L);
	GVL.fbLogger.AddItem (itfItem := GVL_Variable.fbComponent_2_L);
	GVL.fbLogger.AddItem (itfItem := GVL_Variable.fbComponent_3_L);
	
//dodać testowanie dodawania FB_Control FB_Group i FB_Top	
	TcUnit.TEST_FINISHED ();
END_IF
END_METHOD

END_FUNCTION_BLOCK

// ---- POUs/A5_ControlElement_1/FB_ControlElement_HMI_1.TcPOU
FUNCTION_BLOCK FB_ControlElement_HMI_1 EXTENDS FB_BaseControlElement_HMI IMPLEMENTS ITF_ControlElement_HMI_1
VAR
	itfControlElementConnector			: ITF_ControlElement_HMI_Connector_1;
	refstControlElementData				: REFERENCE TO ST_ControlElement_HMI_1;
	
	itfComponent1						: ITF_Component_HMI;
	itfComponent2						: ITF_Component_HMI;
END_VAR

METHOD FB_init : BOOL
VAR_INPUT
	bInitRetains : BOOL; // if TRUE, the retain variables are initialized (warm start / cold start)
	bInCopyCode : BOOL;  // if TRUE, the instance afterwards gets moved into the copy code (online change)
	itfBaseLoggerConnector				: ITF_BaseLogger_HMI_Connector;	//bezpośredni łącznik do logera
	itfControlElementConnector			: ITF_ControlElement_HMI_Init;
	itfComponent1						: ITF_Component_HMI;
	itfComponent2						: ITF_Component_HMI;
END_VAR
//Przypisanie do elementu który własnie stworzyliśmy
THIS^.itfControlElementConnector		:= itfControlElementConnector;
//Przypisanie do elementów z biblioteki
THIS^.itfBaseLoggerElementConnector		:= itfControlElementConnector;
THIS^.itfBaseComponentConnector			:= itfControlElementConnector;
THIS^.itfBaseControlElementConnector	:= itfControlElementConnector;
//
THIS^.itfBaseLoggerConnector			:= itfBaseLoggerConnector;
//
THIS^.itfComponent1						:= itfComponent1;
THIS^.AddComponent (itfComponentHMI		:= itfComponent1);
THIS^.itfComponent2						:= itfComponent2;
this^.AddComponent (itfComponentHMI		:= itfComponent2);

IF (THIS^.itfControlElementConnector <> 0 AND
	THIS^.itfBaseLoggerElementConnector <> 0 AND
	THIS^.itfBaseComponentConnector	<> 0 AND
	THIS^.itfBaseControlElementConnector <> 0 AND
	THIS^.itfBaseLoggerConnector <> 0) THEN
	THIS^.bIsInit						:= TRUE;
END_IF
END_METHOD

METHOD LinkControlElementData : BOOL
VAR_INPUT
	stData				: reference to ST_ControlElement_HMI_Link;
END_VAR
THIS^.refstControlElementData			REF= stData.stControlElement;	//ta zmienna powstaje w elemencie 

THIS^.refstBaseLoggerElementDataHMI		REF= stData.stBaseLoggerElement;	//zmienne z biblioteki ale dopiero tu je moge przypisać 
THIS^.refstBaseComponentDataHMI			REF= stData.stBaseComponent;
THIS^.refstBaseControlElementDataHMI	REF= stData.stBaseControlElement;

THIS^.itfComponent1.LinkComponentData (stData := stData.stComponent1);	//przekazanie danych do elementu podrzędnego np do czujnika
THIS^.itfComponent2.LinkComponentData (stData := stData.stComponent2);

THIS^.CreateLinkToEventsMemory ();	//wywołanie metody linkującą poamięc zgłoszęń

IF (__ISVALIDREF (THIS^.refstControlElementData) AND this^.IsLinkedReferences ()) THEN
	THIS^.bIsValidData		:= TRUE;
	LinkControlElementData	:= TRUE;
END_IF
END_METHOD

END_FUNCTION_BLOCK

// ---- POUs/FB_CreateTepletate1.TcPOU
FUNCTION_BLOCK FB_CreateTepletate1 EXTENDS FB_Base IMPLEMENTS ITF_BaseCreateTemplateOfRecipe
VAR
END_VAR

METHOD CreateTamplateOfRecipe : BOOL
VAR_INPUT
	itfRecipe				: ITF_BaseCreatingTemplateMethod;	//interfejs do obsługi receptur
END_VAR
VAR
	sttmpSkladnik			: ST_BaseDescriptor;
	uiNumberOfTeplates		: UINT;
END_VAR
//	utworzenie szablonu z podaną nazwą
THIS^.SetText (eLocation := E_BaseLocation.pl, wsDescription := "Nazwa szablonu PL");
THIS^.SetText (eLocation := E_BaseLocation.en, wsDescription := "Nazwa szablonu EN");
THIS^.SetText (eLocation := E_BaseLocation.de, wsDescription := "Nazwa szablonu DE");
itfRecipe.AddTemplate (stTexts	:= GVL.fbRecipe.GetTexts ());
uiNumberOfTeplates	:= itfRecipe.GetNumberOfTemplate ();

THIS^.SetTextIn (stIN := sttmpSkladnik, eLocation := E_BaseLocation.pl, wsDescription := "Nazwa skladnika 1 PL");
THIS^.SetTextIn (stIN := sttmpSkladnik, eLocation := E_BaseLocation.en, wsDescription := "Nazwa skladnika 1 EN");
THIS^.SetTextIn (stIN := sttmpSkladnik, eLocation := E_BaseLocation.de, wsDescription := "Nazwa skladnika 1 DE");
THIS^.SetMaxIn (stIN := sttmpSkladnik, rMax := 10000);
THIS^.SetMinIn (stIN := sttmpSkladnik, rMin := 1);
THIS^.SetValueIn (stIN := sttmpSkladnik, rValue := 1111);
THIS^.SetDefaultValueIn (stIN := sttmpSkladnik, rDefaultValue := 1111);
THIS^.SetUnitIn (stIN := sttmpSkladnik, sUnit := 'mm');
itfRecipe.AddIngredientToTemplate (uiNumber := uiNumberOfTeplates, stIngredient := sttmpSkladnik);

THIS^.SetTextIn (stIN := sttmpSkladnik, eLocation := E_BaseLocation.pl, wsDescription := "Nazwa skladnika 2 PL");
THIS^.SetTextIn (stIN := sttmpSkladnik, eLocation := E_BaseLocation.en, wsDescription := "Nazwa skladnika 2 EN");
THIS^.SetTextIn (stIN := sttmpSkladnik, eLocation := E_BaseLocation.de, wsDescription := "Nazwa skladnika 2 DE");
THIS^.SetMaxIn (stIN := sttmpSkladnik, rMax := 10000);
THIS^.SetMinIn (stIN := sttmpSkladnik, rMin := 1);
THIS^.SetValueIn (stIN := sttmpSkladnik, rValue := 1112);
THIS^.SetDefaultValueIn (stIN := sttmpSkladnik, rDefaultValue := 1112);
THIS^.SetUnitIn (stIN := sttmpSkladnik, sUnit := 'mm/s');
itfRecipe.AddIngredientToTemplate (uiNumber := uiNumberOfTeplates, stIngredient := sttmpSkladnik);

THIS^.SetTextIn (stIN := sttmpSkladnik, eLocation := E_BaseLocation.pl, wsDescription := "Nazwa skladnika 3 PL");
THIS^.SetTextIn (stIN := sttmpSkladnik, eLocation := E_BaseLocation.en, wsDescription := "Nazwa skladnika 3 EN");
THIS^.SetTextIn (stIN := sttmpSkladnik, eLocation := E_BaseLocation.de, wsDescription := "Nazwa skladnika 3 DE");
THIS^.SetMaxIn (stIN := sttmpSkladnik, rMax := 10000);
THIS^.SetMinIn (stIN := sttmpSkladnik, rMin := 1);
THIS^.SetValueIn (stIN := sttmpSkladnik, rValue := 1113);
THIS^.SetDefaultValueIn (stIN := sttmpSkladnik, rDefaultValue := 1113);
THIS^.SetUnitIn (stIN := sttmpSkladnik, sUnit := 'ms');
itfRecipe.AddIngredientToTemplate (uiNumber := uiNumberOfTeplates, stIngredient := sttmpSkladnik);
END_METHOD

END_FUNCTION_BLOCK

// ---- POUs/FB_CreateTepletate2.TcPOU
FUNCTION_BLOCK FB_CreateTepletate2 EXTENDS FB_Base IMPLEMENTS ITF_BaseCreateTemplateOfRecipe
VAR
END_VAR

METHOD CreateTamplateOfRecipe : BOOL
VAR_INPUT
	itfRecipe				: ITF_BaseCreatingTemplateMethod;	//interfejs do obsługi receptur
END_VAR
VAR
	sttmpSkladnik			: ST_BaseDescriptor;
	uiNumberOfTeplates		: UINT;
END_VAR
THIS^.SetText (eLocation := E_BaseLocation.pl, wsDescription := "Nazwa szablonu 2 PL");
THIS^.SetText (eLocation := E_BaseLocation.en, wsDescription := "Nazwa szablonu 2 EN");
THIS^.SetText (eLocation := E_BaseLocation.de, wsDescription := "Nazwa szablonu 2 DE");
itfRecipe.AddTemplate (stTexts	:= GVL.fbRecipe.GetTexts ());
uiNumberOfTeplates	:= itfRecipe.GetNumberOfTemplate ();

THIS^.SetTextIn (stIN := sttmpSkladnik, eLocation := E_BaseLocation.pl, wsDescription := "Nazwa skladnika 1 PL");
THIS^.SetTextIn (stIN := sttmpSkladnik, eLocation := E_BaseLocation.en, wsDescription := "Nazwa skladnika 1 EN");
THIS^.SetTextIn (stIN := sttmpSkladnik, eLocation := E_BaseLocation.de, wsDescription := "Nazwa skladnika 1 DE");
THIS^.SetMaxIn (stIN := sttmpSkladnik, rMax := 10000);
THIS^.SetMinIn (stIN := sttmpSkladnik, rMin := 1);
THIS^.SetValueIn (stIN := sttmpSkladnik, rValue := 1111);
THIS^.SetDefaultValueIn (stIN := sttmpSkladnik, rDefaultValue := 1111);
THIS^.SetUnitIn (stIN := sttmpSkladnik, sUnit := 'mm');
itfRecipe.AddIngredientToTemplate (uiNumber := uiNumberOfTeplates, stIngredient := sttmpSkladnik);
END_METHOD

END_FUNCTION_BLOCK
